TYPE Request :
STRUCT
	Command			:UINT;		// Value according to the command table
	Data			:ARRAY[0..18] OF UINT := [0];		
END_STRUCT
END_TYPE

(* stored: Version 1.1.0.1
   DUT Request: Id {7d598dec-a8ba-419b-8579-78edb44d2f5b} *)
